TYPE EntrySearch  :
STRUCT
    ID : LINT;
END_STRUCT
END_TYPE

(* stored: Version 1.1.0.1, ProductVersion 3.1.4024.16
   DUT EntrySearch: Id {d34ca8cc-4398-474b-8b07-a46ed98b6d97} *)
